// Mitsubishi GX Works2 project: 타이머실습1   PLC: Q03UDV

PROGRAM MAIN
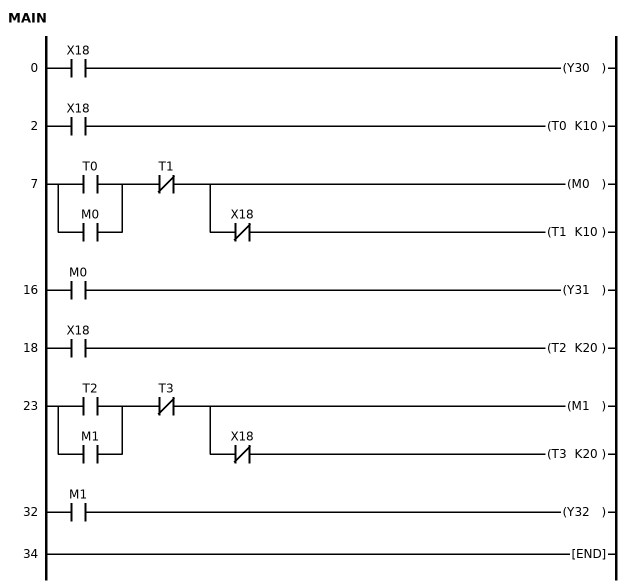
0     LD      X18
      OUT     Y30
2     LD      X18
      OUT     T0 K10
7     LD      T0
      OR      M0
      ANI     T1
      OUT     M0
      ANI     X18
      OUT     T1 K10
16    LD      M0
      OUT     Y31
18    LD      X18
      OUT     T2 K20
23    LD      T2
      OR      M1
      ANI     T3
      OUT     M1
      ANI     X18
      OUT     T3 K20
32    LD      M1
      OUT     Y32
34    END
END_PROGRAM
